FUNCTION_BLOCK FB_NullLogger IMPLEMENTS I_Logger				// Null logger implementation

METHOD PUBLIC debug : BOOL	// Logs the data with log level 'DEBUG'
VAR_INPUT
	iData:		T_DEFAULT_STR;						// Data to be logged, limited to 255 characters
END_VAR
// Do nothing
END_METHOD

METHOD PUBLIC deregister : BOOL
VAR_INPUT
	iWho:				T_SHORT_STR;
END_VAR
END_METHOD

METHOD PUBLIC doLog : BOOL
VAR_INPUT
	iData:		T_DEFAULT_STR;						// Data to be logged, limited to 255 characters
	iLevel:		E_LOG_LEVEL := E_LOG_LEVEL.ERROR;	// Log level
END_VAR
END_METHOD

METHOD PUBLIC error : BOOL	// Logs the data with log level 'ERROR'
VAR_INPUT
	iData:		T_DEFAULT_STR;						// Data to be logged, limited to 255 characters
END_VAR
// Do nothing
END_METHOD

METHOD PUBLIC info : BOOL	// Logs the data with log level 'INFO'
VAR_INPUT
	iData:		T_DEFAULT_STR;						// Data to be logged, limited to 255 characters
END_VAR
// Do nothing
END_METHOD

METHOD PUBLIC register : BOOL
VAR_INPUT
	iWho:		T_SHORT_STR;
	iObserver:	I_Logger;
END_VAR
END_METHOD

METHOD PUBLIC trace : BOOL	// Logs the data with log level 'TRACE'
VAR_INPUT
	iData:		T_DEFAULT_STR;						// Data to be logged, limited to 255 characters
END_VAR
// Do nothing
END_METHOD

METHOD PUBLIC warn : BOOL	// Logs the data with log level 'WARN'
VAR_INPUT
	iData:		T_DEFAULT_STR;						// Data to be logged, limited to 255 characters
END_VAR
// Do nothing
END_METHOD

END_FUNCTION_BLOCK

(* stored: Version 1.1.0.1, ProductVersion 3.1.4026.18
   POU FB_NullLogger: Id {eeeff7f9-3eb4-4f89-96d0-1cc044d80d00}, SpecialFunc None
   Method debug: Id {251af618-dcc2-4891-a05d-135b0a346a28}
   Method deregister: Id {f3d80110-5c64-4f37-bbde-87868de5e4b5}
   Method doLog: Id {4e979eaf-b7b4-49b8-a400-47aa0e342525}
   Method error: Id {43f9d53c-7213-48e4-8bb8-91059cc72413}
   Method info: Id {2b677cbc-5e14-4ced-90b6-4591d73d5d6f}
   Method register: Id {7f5445c7-7066-4067-9d52-634e7a0bcfa0}
   Method trace: Id {b8d908ce-1427-4843-8fc6-835a04e23249}
   Method warn: Id {bcbec991-2ee8-4559-bf67-31e28066da99} *)
